GLOBALCONSTANTS HandshakeConst (* Handshake pattern demo constants *)
  (* Standard: 61499-1; Description: Copyright (c) 2026 Meisterschulen am Ostbahnhof This program and the accompanying materials are made available under the terms of the Eclipse Public License 2.0 which is available at https://www.eclipse.org/legal/epl-2.0/ SPDX-License-Identifier: EPL-2.0 *)
  (* Version 1.0, 2026-08-31, Franz Höpfinger, Meisterschulen am Ostbahnhof, Handshake design pattern (IEC 61499 primer course, Module 6, Valeriy Vyatkin), demo constants for the WSTRING variant *)
  PACKAGE Meins::DesingPatterns::HandshakePattern::const;
  VAR_GLOBAL CONSTANT
    ACK_PAYLOAD : WSTRING := "ack"; (* Fixed acknowledgement payload used by the WSTRING Handshake demo (Responder's CNF, Requester's RSP) *)
  END_VAR
END_GLOBALCONSTANTS
